INTERFACE IPAScaleGravimetric EXTENDS IPAScale

END_INTERFACE

(* stored: Version 1.1.0.1, ProductVersion 3.1.4020.12
   Itf IPAScaleGravimetric: Id {ba942767-991c-4d51-bd8d-b46eb8f07034} *)
